(* PLC project conveyor_belt, Dassault Systèmes ControlBuild 2024x *)
(* stored: creationDateTime 2023-10-03T11:12:58-01:00 *)

(* This module simulates the behaviour of a conveyor-belt driven by an analog value of the speed. *)
FUNCTION_BLOCK equipment_library.conveyor_belt
  VAR_INPUT
    volumeIn : REAL := 0.0;
    depositPosition : REAL := 0.0;
    speed : REAL := 0.0;
    openValve : BOOL := false;
  END_VAR
  VAR_OUTPUT
    volumeOutFwd : REAL := 0.0;
    volumeOutBwd : REAL := 0.0;
    controllerRot : BOOL := false;
    volumeOutValve : REAL := 0.0;
  END_VAR
  VAR
    materialHead : REAL := 0.0;
    materialTailEnd : REAL := 0.0;
    deviation : REAL := 0.0;
    volumeOn : REAL := 0.0;
    increment : REAL := 0.0;
    effectiveLength : REAL := 0.0;
    valvePassage : BOOL := false;
  END_VAR
  VAR CONSTANT
    controllerLogic : BOOL := true;
    conveyorLength : REAL := 20.0;
    controllerRotThres : REAL := 50.0;
    ratedSpeed : REAL := 1.0;
    weighingPosition : REAL := 5.0;
    valvePosition : REAL := 10.0;
  END_VAR
  VAR
    d_sticking : BOOL := false;
    v_d_sticking : BOOL := false;
  END_VAR


ACTION C_source_code:
/* -----------------------------------------------------------------	*/
/* Type : Model of Operative Behaviour					*/
/* Catégorie :   batch							*/
/* Author : Dassault Systemes						*/
/* Update date : June 2018							*/
/* -----------------------------------------------------------------	*/
/* This module simulates the bahaviour of a conveyor-belt driven by	*/
/* an analog value of the speed.             				*/
/* ----------------------------------------------------------------	*/


/* Real variables of type 'double' are used for best accuracy		*/
double head=0.0;	/* Position of material's head   		     	*/
double tailEnd=0.0;	/* Position of material's tail end 		*/
double incr=0.0;	/* Increment of position for head and/or tail end	*/
double diff=0.0;	/* Length of material ejected by the conveyor-belt	*/

head = materialHead;
tailEnd = materialTailEnd;

/* Manage the rotation controller						*/
/* ----------------------------------------------------------------	*/
if (d_sticking) controllerRot = v_d_sticking;
else
	controllerRot = (fabs(speed) >= controllerRotThres) ^ !controllerLogic;



/* Compute the position of material's ejection				*/
/* ----------------------------------------------------------------	*/
valvePassage=0;

if(openValve) {
	if (speed>0.0)
	{
		effectiveLength=fabs(depositPosition - conveyorLength);
		if (valvePosition>=depositPosition)	
		{
			effectiveLength=fabs(depositPosition - valvePosition);
			valvePassage=1;
		}
	}
	else
	{
		effectiveLength=depositPosition;
		if (valvePosition<=depositPosition)	
		{
			effectiveLength=fabs(depositPosition - valvePosition);
			valvePassage=1;
		}
	}
}
else {
	if (speed>= 0.0) effectiveLength=fabs(depositPosition - conveyorLength);
	else effectiveLength= depositPosition;
}

/* Compute the position of material			 		*/
/* ----------------------------------------------------------------	*/

incr = speed * (CLOCK_PERIOD / 1000000);
increment =incr;

if  (volumeOn==0.0) {
       head=tailEnd=depositPosition;
	materialHead = depositPosition;
       materialTailEnd =depositPosition;
}
if((volumeIn==0.0)&& (materialHead!=depositPosition)) {
	head+=incr;
	materialHead=head;
	tailEnd+=incr;
	materialTailEnd = tailEnd;
} 
 else {
 	tailEnd=depositPosition;
	materialTailEnd = depositPosition;
	if ((volumeOn != 0.0) || (volumeIn != 0.0)) head+=incr;
	materialHead=head;         
}



/* Compute the volume of material on the conveyor-belt bande        	*/
/* ----------------------------------------------------------------	*/
if ((materialHead-materialTailEnd !=0) || (speed==0.0))
{
          volumeOn += volumeIn;
}
if (volumeOn < 0.0) volumeOn = 0.0;



/* Compute the volume of material ejected to BWD   			*/
/* ----------------------------------------------------------------	*/
volumeOutBwd = 0.0;
volumeOutValve=0.0;
if ((speed<0.0) && (head<0.0) && !valvePassage) {
	diff = fabs(head);
              
	if (fabs(tailEnd - head) > 0.0) {
		volumeOutBwd= diff * volumeOn/ fabs(tailEnd - head);	
	}
	else volumeOutBwd=volumeOn;

	head=head+diff;
	materialHead = head;

}
if ((speed<0.0) && (head <= valvePosition) && valvePassage) {
	diff = -incr;
	if (fabs(tailEnd - head) > 0.0) {
		volumeOutValve= diff * volumeOn/ fabs(tailEnd - head);	
	}
	else volumeOutValve=volumeOn;

	head=head+diff;
	materialHead = head;
}


/* Compute the volume of material ejected to FWD   			*/
/* ----------------------------------------------------------------	*/
volumeOutFwd = 0.0;
if ((speed>0.0) && (fabs(head) > fabs(depositPosition+effectiveLength))) {
	diff = fabs(fabs(head) - fabs(depositPosition+effectiveLength));
	deviation = diff;
	if (diff > 0.0) {
		if(valvePassage) {
			if(fabs(head - tailEnd)>0.0) volumeOutValve = diff * volumeOn /fabs(head - tailEnd);
			else volumeOutValve=volumeOn;
			volumeOutFwd=0.0;
		}
		else {
			if(fabs(head - tailEnd)>0.0) volumeOutFwd = diff * volumeOn /fabs(head - tailEnd);
			else volumeOutFwd=volumeOn;
			volumeOutValve=0.0;
		}
	}
	
	head=head-diff;
	materialHead = head;
}



/* Compute the volume of material on the conveyor   			*/
/* ----------------------------------------------------------------	*/
volumeOn +=  - (volumeOutBwd+volumeOutFwd+volumeOutValve);
END_ACTION

ACTION C_header:
#include<math.h> 	/* pour fonction fabs */
END_ACTION
END_FUNCTION_BLOCK
